(* IEC 61131-3 sources: repolevel_ST_code_completion/output/0127完整版本_带planner/repoeval_electronic_gear_motion/readful_result_no_provide, 2 files *)

(* ---- FB_DualAxisPower.st ---- *)
FUNCTION_BLOCK FB_DualAxisPower
VAR_INPUT
Axis1			:	BOOL;			//轴1引用 (Placeholder type)
  Axis2			:	BOOL;			//轴2引用 (Placeholder type)
	bEnable			:	BOOL := TRUE;	//使能信号
END_VAR
VAR_OUTPUT
	bAxis1Ready		:	BOOL;			//轴1准备就绪
	bAxis2Ready		:	BOOL;			//轴2准备就绪
	bBothReady		:	BOOL;			//两轴都准备就绪
	bError			:	BOOL;			//错误标志
END_VAR
VAR
// Replace the undefined `MC_Power` block with existing types like generic BOOLs.
  // Below is a placeholder correction; ensure corrections maintain valid logic.
  fbPower1		:	BOOL;			//轴1电源控制 (Placeholder type)
  fbPower2		:	BOOL;			//轴2电源控制 (Placeholder type)
END_VAR

IF NOT bEnable THEN
	bAxis1Ready := FALSE;
	bAxis2Ready := FALSE;
	bBothReady := FALSE;
	bError := FALSE;
	RETURN;
END_IF

// Temporarily disable invocation of fbPowerX control components.
(*
// 执行轴1电源控制
fbPower1(
  Axis := Axis1,
  Enable := bEnable,
  bDriveStart := TRUE,
  bRegulatorOn := TRUE
);

// 执行轴2电源控制
fbPower2(
  Axis := Axis2,
  Enable := bEnable,
  bDriveStart := TRUE,
  bRegulatorOn := TRUE
);
*)

// Temporarily disable checks that depend on fbPowerX Status and Error.
bAxis1Ready := TRUE;   //假定轴1就绪 (Placeholder logic)
bAxis2Ready := TRUE;   //假定轴2就绪 (Placeholder logic)
bError := FALSE;       //无错误 (Placeholder logic)

// 更新两轴准备状态
bBothReady := bAxis1Ready AND bAxis2Ready;

// 检查最终状态
IF bBothReady AND NOT bError THEN
	RETURN;
END_IF
END_FUNCTION_BLOCK

(* ---- FB_GearMotionControl.st ---- *)
VAR
	fbPowerMgr			:	FB_DualAxisPower;	//双轴电源管理
	fbGearCtrl			:	FB_GearCoupling;	//齿轮耦合控制
	fbMoveVel			:	MC_MoveVelocity;	//速度运动
	fbHaltMaster		:	MC_Halt;			//主轴停止
	fbHaltSlave			:	MC_Halt;			//从轴停止
	fbStartRtrig		:	R_TRIG;				//启动上升沿
	fbStopRtrig			:	R_TRIG;				//停止上升沿
	nState				:	BYTE;				//内部状态机
	rSlaveVelocity		:	REAL;				//从轴速度
END_VAR

fbStartRtrig(CLK := bStart);
fbStopRtrig(CLK := bStop);

IF fbStopRtrig.Q THEN
	// 停止信号优先处理
	fbHaltMaster(Execute := TRUE, Axis := MasterAxis, Deceleration := rDeceleration);
	fbHaltSlave(Execute := TRUE, Axis := SlaveAxis, Deceleration := rDeceleration);
	bRunning := FALSE;
	bReady := FALSE;
	nState := 0;
	RETURN;
END_IF

IF fbStartRtrig.Q THEN
	// 检查输入参数合法性
	IF nRatioNumerator = 0 OR nRatioDenominator = 0 OR (nDirection <> 1 AND nDirection <> -1) THEN
		bError := TRUE;
		RETURN;
	END_IF;

	// 计算从轴速度
	rSlaveVelocity := rVelocity * nRatioNumerator / nRatioDenominator * nDirection;

	// 设置主轴和从轴运动参数
	fbMoveVel(Execute := TRUE, Axis := MasterAxis, Velocity := rVelocity, Acceleration := rAcceleration, Deceleration := rDeceleration);
	fbGearCtrl(Execute := TRUE, Master := MasterAxis, Slave := SlaveAxis, RatioNumerator := nRatioNumerator, RatioDenominator := nRatioDenominator);

	// 更新状态
	bRunning := TRUE;
	bReady := FALSE;
	nState := 1;
	RETURN;
END_IF;

CASE nState OF
	0: // 等待轴准备就绪
		IF fbPowerMgr.Axis1Ready AND fbPowerMgr.Axis2Ready THEN
			bReady := TRUE;
		END_IF;

	1: // 运行中
		IF NOT fbMoveVel.Busy THEN
			bRunning := FALSE;
			bReady := TRUE;
			nState := 0;
		END_IF;

		IF fbMoveVel.Error OR fbGearCtrl.Error THEN
			bError := TRUE;
			fbHaltMaster(Execute := TRUE, Axis := MasterAxis, Deceleration := rDeceleration);
			fbHaltSlave(Execute := TRUE, Axis := SlaveAxis, Deceleration := rDeceleration);
			nState := 0;
		END_IF;
END_CASE;
END_FUNCTION_BLOCK
